// TIA Portal V19 export
FUNCTION_BLOCK "Losma_FB"   // FB154, LAD
TITLE = MATERIAL LUBRICATION (LOSMA)
// stored: MemoryReserve 100, SetENOAutomatically false
   VAR_INPUT
      AreaInterface : "AreaInterface";
      ZSI : "udt_ZoneSafetyInterface";
      DSI : "udt_DeviceSafetyInterface";
      DataIn : Struct
         PbPumpStop : Bool;
         PbPumpStart : Bool;
         PbBlowerStop : Bool;
         PbBlowerStart : Bool;
         PbOilSeparatorStop : Bool;
         PbOilSeparatorStart : Bool;
         SensorLevelTank : Bool;
         SensorStartCloth : Bool;
         SensorOilSeparator : Bool;
         PumpFdbkRunning : Bool;
         OilSeparatorFdbkRunning : Bool;
         ClothFdbkRunning : Bool;
      END_STRUCT;
      CIn : Struct
         EnableStopInPhase : Bool;
         EnableStopProgrammed : Bool;
         EnableAborting : Bool;
         MaterialMoving : Bool;
      END_STRUCT;
      Config : Struct
         EnableWngSystemOff : Bool;
         ClothExist : Bool;
         OilSeparatorExist : Bool;
         LowTankLevelDly : Time;
      END_STRUCT;
   END_VAR
   VAR_OUTPUT
      MachineInterface : "MachineInterface";
      DataOut : Struct
         KmPump : Bool;
         KmCloth : Bool;
         KmOilSeparator : Bool;
         BlowerSolenoidValve : Bool;
         PumpLamp : Bool;
         BlowerLamp : Bool;
      END_STRUCT;
      COut : Struct
         PumpIsRunning : Bool;
         BlowerIsRunning : Bool;
         OilSeparatorIsRunning : Bool;
      END_STRUCT;
   END_VAR
   VAR_IN_OUT
      PersistentValues : Struct
         Par : Struct
            PumpOnOff : Bool;
            BlowerOnOff : Bool;
            OilSeparator : Bool;
            PumpDelayOff : Time;
            BlowerDelayOff : Time;
         END_STRUCT;
      END_STRUCT;
   END_VAR
   VAR
      Sts : Struct
         AlarmsPresence : Bool;
         WarningsPresence : Bool;
         IsStandstill : Bool;
         PumpRunReq : Bool;
         BlowerRunReq : Bool;
         OilSeparatorRunReq : Bool;
         CndPump { ExternalAccessible := 'False'; ExternalVisible := 'False'; ExternalWritable := 'False'} : Bool;
         CndBlower { ExternalAccessible := 'False'; ExternalVisible := 'False'; ExternalWritable := 'False'} : Bool;
         CndCloth { ExternalAccessible := 'False'; ExternalVisible := 'False'; ExternalWritable := 'False'} : Bool;
         CndOilSeparator : Bool;
      END_STRUCT;
      Ctrl : Struct
         RstAlarms : Bool;
         StopDueDoorOpeningRequest : Bool;
         SafeStop : Bool;
         StopInPhase : Bool;
         StopProgrammed : Bool;
         Pump_ManStart : Bool;
         Pump_AutStart : Bool;
         Blower_ManStart : Bool;
         Blower_AutStart : Bool;
         Cloth_AutStart : Bool;
         OilSeparator_ManStart : Bool;
         OilSeparator_AutStart : Bool;
      END_STRUCT;
      Alr : Struct
         LowTankLevel : Bool;
         HighLevelOilTank : Bool;
         Pump : "MotorAlr";
         Cloth : "MotorAlr";
         OilSeparator : "MotorAlr";
      END_STRUCT;
      Wng : Struct
         NoAutReady : Bool;
         PumpOff : Bool;
         BlowerOff : Bool;
         OilSeparatorOff : Bool;
      END_STRUCT;
      M_Pump : "Motor";
      M_Cloth : "Motor";
      M_OilSeparator : "Motor";
      TON_DelayBlowerStop : IEC_TIMER;
      TON_DelayPumpStop : IEC_TIMER;
      TON_LowTankLevel : IEC_TIMER;
      TON_DelayNoPendingCmd : IEC_TIMER;
      TON_OilTankLevelIsFull : IEC_TIMER;
      PbPumpStart_PEAux : Bool;
      PbBlowerStart_PEAux : Bool;
      PbOilSeparatorStart_PEAux : Bool;
   END_VAR
   VAR_TEMP   // added for the SCL form of the ladder/FBD networks
      _w1 : Bool;
   END_VAR
BEGIN

REGION Network 1 (SCL): Reset alarms command
   #Ctrl.RstAlarms := #AreaInterface.RstAlarms;

   IF  #Ctrl.RstAlarms THEN
       #Wng.NoAutReady := FALSE;
       #Alr.LowTankLevel := FALSE;
       #Alr.HighLevelOilTank := FALSE;
   END_IF;
END_REGION

REGION Network 2: Warning Pump / Blower off
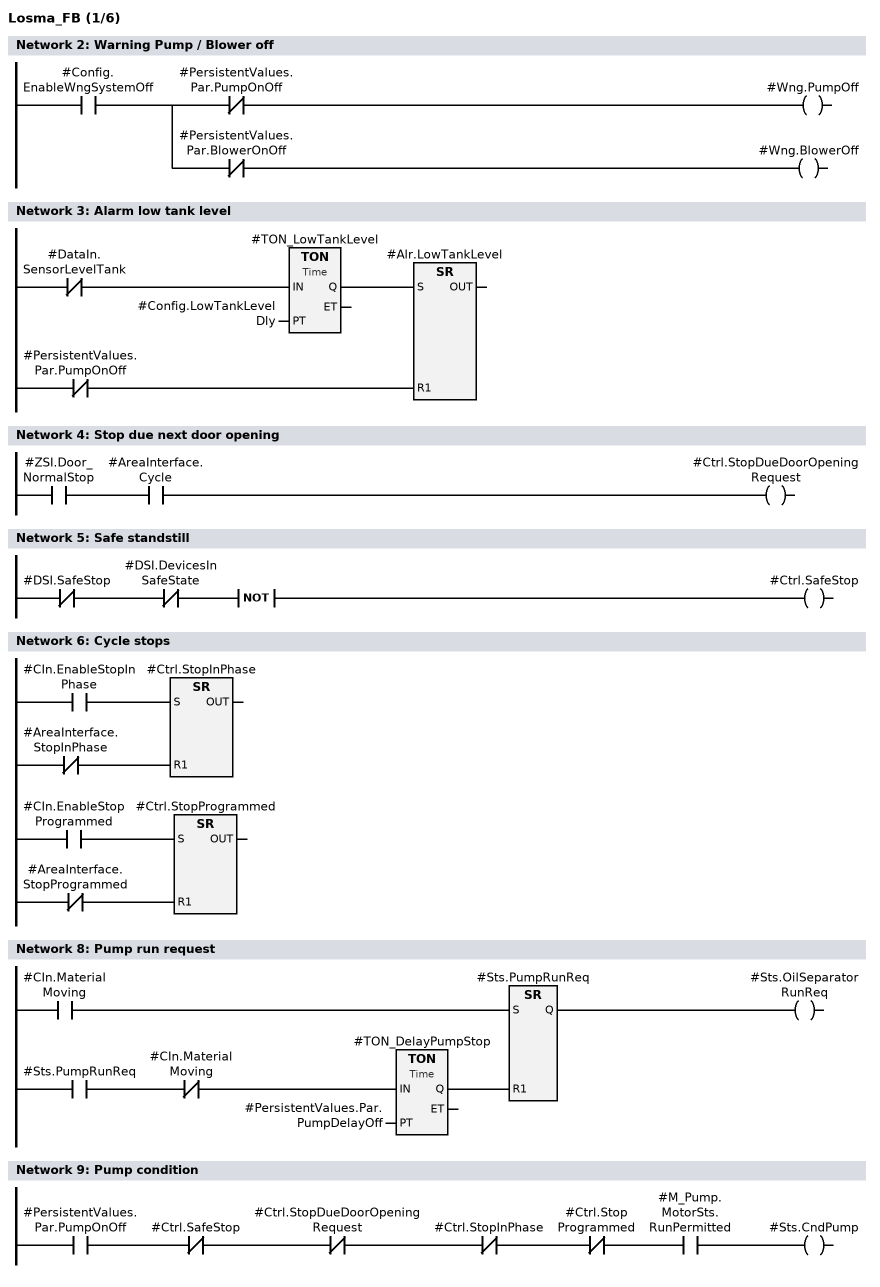
   RUNG wire#powerrail
      Contact( #Config.EnableWngSystemOff )
      wire#w1
      I_Contact( #PersistentValues.Par.PumpOnOff )
      Coil( #Wng.PumpOff )
   END_RUNG
   RUNG wire#w1
      I_Contact( #PersistentValues.Par.BlowerOnOff )
      Coil( #Wng.BlowerOff )
   END_RUNG
   // the same network as SCL:
   #Wng.PumpOff := #Config.EnableWngSystemOff AND NOT #PersistentValues.Par.PumpOnOff;
   #Wng.BlowerOff := #Config.EnableWngSystemOff AND NOT #PersistentValues.Par.BlowerOnOff;
END_REGION

REGION Network 3: Alarm low tank level
   RUNG wire#powerrail
      I_Contact( #DataIn.SensorLevelTank )
      { S7_Templates := "time_type := Time" } #TON_LowTankLevel.TON(pt := #Config.LowTankLevelDly, et =>)
      S_SR(operand := #Alr.LowTankLevel, r1 := wire#w1)
   END_RUNG
   RUNG wire#powerrail
      I_Contact( #PersistentValues.Par.PumpOnOff )
   END_RUNG wire#w1
   // the same network as SCL:
   #TON_LowTankLevel.TON(IN := NOT #DataIn.SensorLevelTank, PT := #Config.LowTankLevelDly);
   IF #TON_LowTankLevel.Q THEN
       #Alr.LowTankLevel := TRUE;   // SR flip-flop
   END_IF;
   IF NOT #PersistentValues.Par.PumpOnOff THEN #Alr.LowTankLevel := FALSE; END_IF;
END_REGION

REGION Network 4: Stop due next door opening
   RUNG wire#powerrail
      Contact( #ZSI.Door_NormalStop )
      Contact( #AreaInterface.Cycle )
      Coil( #Ctrl.StopDueDoorOpeningRequest )
   END_RUNG
   // the same network as SCL:
   #Ctrl.StopDueDoorOpeningRequest := #ZSI.Door_NormalStop AND #AreaInterface.Cycle;
END_REGION

REGION Network 5: Safe standstill
   RUNG wire#powerrail
      I_Contact( #DSI.SafeStop )
      I_Contact( #DSI.DevicesInSafeState )
      Not()
      Coil( #Ctrl.SafeStop )
   END_RUNG
   // the same network as SCL:
   #Ctrl.SafeStop := NOT (NOT #DSI.SafeStop AND NOT #DSI.DevicesInSafeState);
END_REGION

REGION Network 6: Cycle stops
   RUNG wire#powerrail
      Contact( #CIn.EnableStopInPhase )
      S_SR(operand := #Ctrl.StopInPhase, r1 := wire#w1)
   END_RUNG
   RUNG wire#powerrail
      I_Contact( #AreaInterface.StopInPhase )
   END_RUNG wire#w1
   RUNG wire#powerrail
      Contact( #CIn.EnableStopProgrammed )
      S_SR(operand := #Ctrl.StopProgrammed, r1 := wire#w2)
   END_RUNG
   RUNG wire#powerrail
      I_Contact( #AreaInterface.StopProgrammed )
   END_RUNG wire#w2
   // the same network as SCL:
   IF #CIn.EnableStopInPhase THEN
       #Ctrl.StopInPhase := TRUE;   // SR flip-flop
   END_IF;
   IF NOT #AreaInterface.StopInPhase THEN #Ctrl.StopInPhase := FALSE; END_IF;
   IF #CIn.EnableStopProgrammed THEN
       #Ctrl.StopProgrammed := TRUE;   // SR flip-flop
   END_IF;
   IF NOT #AreaInterface.StopProgrammed THEN #Ctrl.StopProgrammed := FALSE; END_IF;
END_REGION

REGION Network 7: <<< PUMP >>>
END_REGION

REGION Network 8: Pump run request
   RUNG wire#powerrail
      Contact( #CIn.MaterialMoving )
      S_SR(operand := #Sts.PumpRunReq, r1 := wire#w1)
      Coil( #Sts.OilSeparatorRunReq )
   END_RUNG
   RUNG wire#powerrail
      Contact( #Sts.PumpRunReq )
      I_Contact( #CIn.MaterialMoving )
      { S7_Templates := "time_type := Time" } #TON_DelayPumpStop.TON(pt := #PersistentValues.Par.PumpDelayOff, et =>)
   END_RUNG wire#w1
   // the same network as SCL:
   #TON_DelayPumpStop.TON(IN := #Sts.PumpRunReq AND NOT #CIn.MaterialMoving,
                          PT := #PersistentValues.Par.PumpDelayOff);
   IF #CIn.MaterialMoving THEN
       #Sts.PumpRunReq := TRUE;   // SR flip-flop
   END_IF;
   IF #TON_DelayPumpStop.Q THEN #Sts.PumpRunReq := FALSE; END_IF;
   #Sts.OilSeparatorRunReq := #Sts.PumpRunReq;
END_REGION

REGION Network 9: Pump condition
   RUNG wire#powerrail
      Contact( #PersistentValues.Par.PumpOnOff )
      I_Contact( #Ctrl.SafeStop )
      I_Contact( #Ctrl.StopDueDoorOpeningRequest )
      I_Contact( #Ctrl.StopInPhase )
      I_Contact( #Ctrl.StopProgrammed )
      Contact( #M_Pump.MotorSts.RunPermitted )
      Coil( #Sts.CndPump )
   END_RUNG
   // the same network as SCL:
   #Sts.CndPump := #PersistentValues.Par.PumpOnOff AND NOT #Ctrl.SafeStop AND NOT #Ctrl.StopDueDoorOpeningRequest AND NOT #Ctrl.StopInPhase AND NOT #Ctrl.StopProgrammed AND #M_Pump.MotorSts.RunPermitted;
END_REGION

REGION Network 10: Pump automatic start
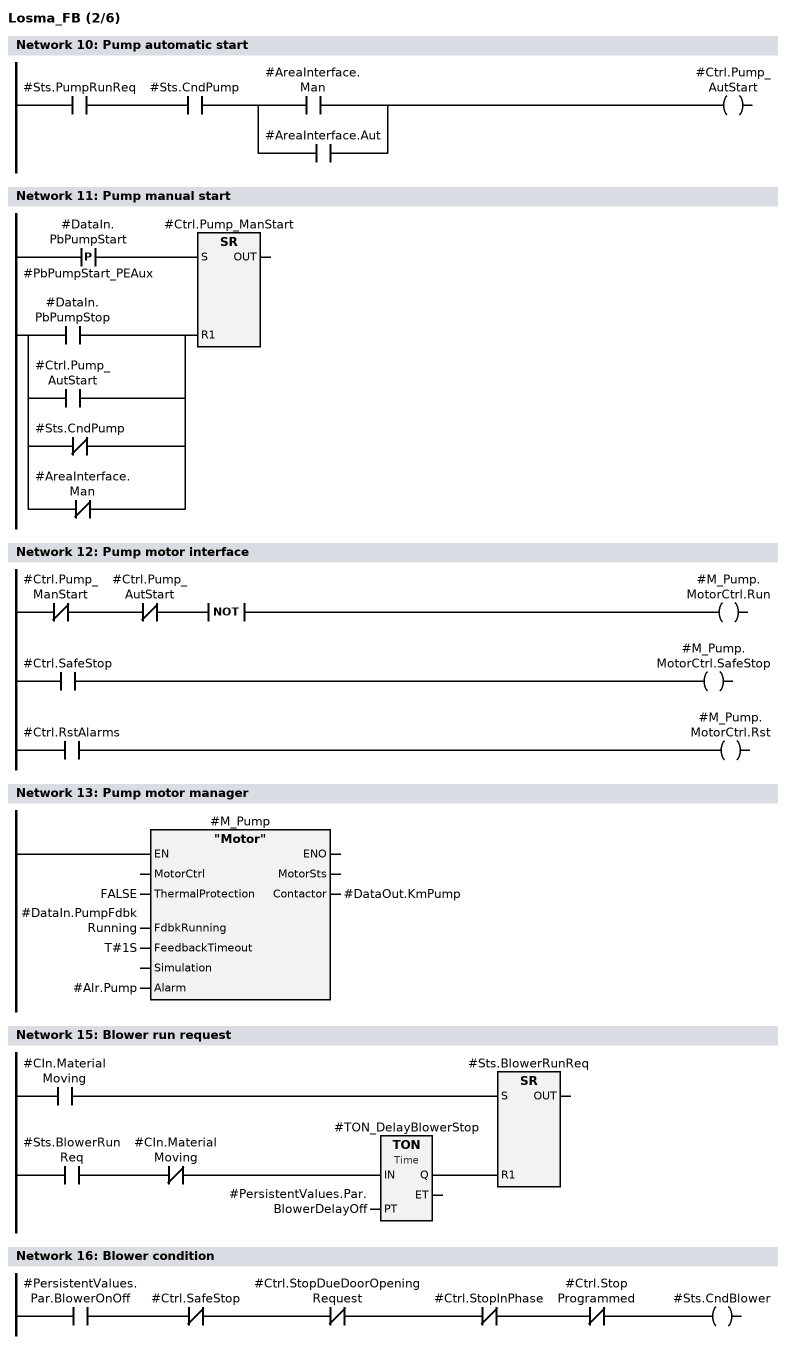
   RUNG wire#powerrail
      Contact( #Sts.PumpRunReq )
      Contact( #Sts.CndPump )
      wire#w1
      Contact( #AreaInterface.Man )
      wire#w2
      Coil( #Ctrl.Pump_AutStart )
   END_RUNG
   RUNG wire#w1
      Contact( #AreaInterface.Aut )
   END_RUNG wire#w2
   // the same network as SCL:
   #Ctrl.Pump_AutStart := #Sts.PumpRunReq AND #Sts.CndPump AND (#AreaInterface.Man OR #AreaInterface.Aut);
END_REGION

REGION Network 11: Pump manual start
   RUNG wire#powerrail
      P_Contact(operand := #DataIn.PbPumpStart, bit := #PbPumpStart_PEAux)
      S_SR(operand := #Ctrl.Pump_ManStart, r1 := wire#w1)
   END_RUNG
   RUNG wire#powerrail
      Contact( #DataIn.PbPumpStop )
   END_RUNG wire#w1
   RUNG wire#powerrail
      Contact( #Ctrl.Pump_AutStart )
   END_RUNG wire#w1
   RUNG wire#powerrail
      I_Contact( #Sts.CndPump )
   END_RUNG wire#w1
   RUNG wire#powerrail
      I_Contact( #AreaInterface.Man )
   END_RUNG wire#w1
   // the same network as SCL:
   #_w1 := #DataIn.PbPumpStart AND NOT #PbPumpStart_PEAux;   // rising edge of #DataIn.PbPumpStart
   #PbPumpStart_PEAux := #DataIn.PbPumpStart;
   IF #_w1 THEN
       #Ctrl.Pump_ManStart := TRUE;   // SR flip-flop
   END_IF;
   IF #DataIn.PbPumpStop OR #Ctrl.Pump_AutStart OR NOT #Sts.CndPump OR NOT #AreaInterface.Man THEN
       #Ctrl.Pump_ManStart := FALSE;
   END_IF;
END_REGION

REGION Network 12: Pump motor interface
   RUNG wire#powerrail
      I_Contact( #Ctrl.Pump_ManStart )
      I_Contact( #Ctrl.Pump_AutStart )
      Not()
      Coil( #M_Pump.MotorCtrl.Run )
   END_RUNG
   RUNG wire#powerrail
      Contact( #Ctrl.SafeStop )
      Coil( #M_Pump.MotorCtrl.SafeStop )
   END_RUNG
   RUNG wire#powerrail
      Contact( #Ctrl.RstAlarms )
      Coil( #M_Pump.MotorCtrl.Rst )
   END_RUNG
   // the same network as SCL:
   #M_Pump.MotorCtrl.Run := NOT (NOT #Ctrl.Pump_ManStart AND NOT #Ctrl.Pump_AutStart);
   #M_Pump.MotorCtrl.SafeStop := #Ctrl.SafeStop;
   #M_Pump.MotorCtrl.Rst := #Ctrl.RstAlarms;
END_REGION

REGION Network 13: Pump motor manager
   RUNG wire#powerrail
      #M_Pump(MotorCtrl :=, ThermalProtection := FALSE, FdbkRunning := #DataIn.PumpFdbkRunning, FeedbackTimeout := T#1S, Simulation :=, Alarm := #Alr.Pump, MotorSts =>, Contactor => #DataOut.KmPump)
   END_RUNG
   // the same network as SCL:
   #M_Pump(ThermalProtection := FALSE,   // "Motor"
           FdbkRunning := #DataIn.PumpFdbkRunning,
           FeedbackTimeout := T#1S,
           Alarm := #Alr.Pump,
           Contactor => #DataOut.KmPump);
END_REGION

REGION Network 14: <<< BLOWER >>>
END_REGION

REGION Network 15: Blower run request
   RUNG wire#powerrail
      Contact( #CIn.MaterialMoving )
      S_SR(operand := #Sts.BlowerRunReq, r1 := wire#w1)
   END_RUNG
   RUNG wire#powerrail
      Contact( #Sts.BlowerRunReq )
      I_Contact( #CIn.MaterialMoving )
      { S7_Templates := "time_type := Time" } #TON_DelayBlowerStop.TON(pt := #PersistentValues.Par.BlowerDelayOff, et =>)
   END_RUNG wire#w1
   // the same network as SCL:
   #TON_DelayBlowerStop.TON(IN := #Sts.BlowerRunReq AND NOT #CIn.MaterialMoving,
                           PT := #PersistentValues.Par.BlowerDelayOff);
   IF #CIn.MaterialMoving THEN
       #Sts.BlowerRunReq := TRUE;   // SR flip-flop
   END_IF;
   IF #TON_DelayBlowerStop.Q THEN #Sts.BlowerRunReq := FALSE; END_IF;
END_REGION

REGION Network 16: Blower condition
   RUNG wire#powerrail
      Contact( #PersistentValues.Par.BlowerOnOff )
      I_Contact( #Ctrl.SafeStop )
      I_Contact( #Ctrl.StopDueDoorOpeningRequest )
      I_Contact( #Ctrl.StopInPhase )
      I_Contact( #Ctrl.StopProgrammed )
      Coil( #Sts.CndBlower )
   END_RUNG
   // the same network as SCL:
   #Sts.CndBlower := #PersistentValues.Par.BlowerOnOff AND NOT #Ctrl.SafeStop AND NOT #Ctrl.StopDueDoorOpeningRequest AND NOT #Ctrl.StopInPhase AND NOT #Ctrl.StopProgrammed;
END_REGION

REGION Network 17: Blower automatc start / blower automatc start
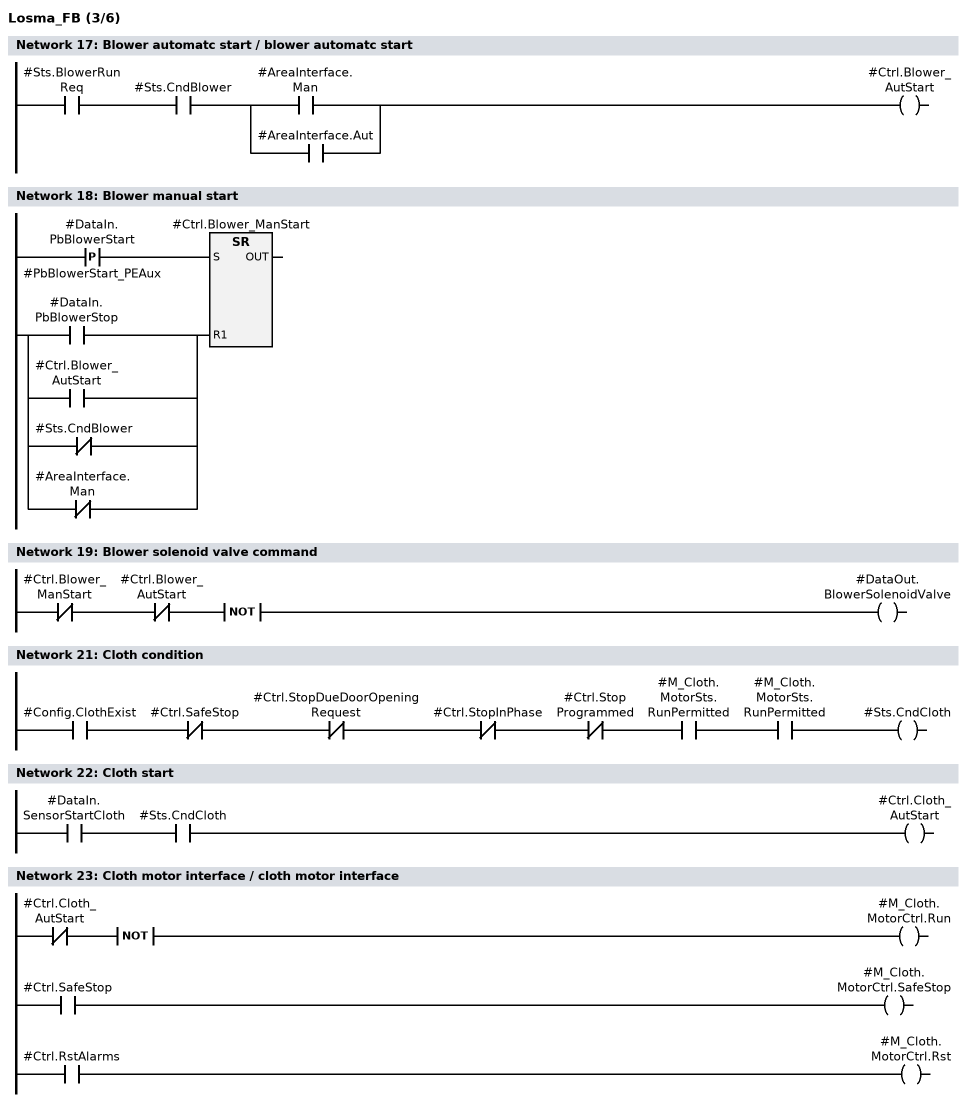
   RUNG wire#powerrail
      Contact( #Sts.BlowerRunReq )
      Contact( #Sts.CndBlower )
      wire#w1
      Contact( #AreaInterface.Man )
      wire#w2
      Coil( #Ctrl.Blower_AutStart )
   END_RUNG
   RUNG wire#w1
      Contact( #AreaInterface.Aut )
   END_RUNG wire#w2
   // the same network as SCL:
   #Ctrl.Blower_AutStart := #Sts.BlowerRunReq AND #Sts.CndBlower AND (#AreaInterface.Man OR #AreaInterface.Aut);
END_REGION

REGION Network 18: Blower manual start
   RUNG wire#powerrail
      P_Contact(operand := #DataIn.PbBlowerStart, bit := #PbBlowerStart_PEAux)
      S_SR(operand := #Ctrl.Blower_ManStart, r1 := wire#w1)
   END_RUNG
   RUNG wire#powerrail
      Contact( #DataIn.PbBlowerStop )
   END_RUNG wire#w1
   RUNG wire#powerrail
      Contact( #Ctrl.Blower_AutStart )
   END_RUNG wire#w1
   RUNG wire#powerrail
      I_Contact( #Sts.CndBlower )
   END_RUNG wire#w1
   RUNG wire#powerrail
      I_Contact( #AreaInterface.Man )
   END_RUNG wire#w1
   // the same network as SCL:
   #_w1 := #DataIn.PbBlowerStart AND NOT #PbBlowerStart_PEAux;   // rising edge of #DataIn.PbBlowerStart
   #PbBlowerStart_PEAux := #DataIn.PbBlowerStart;
   IF #_w1 THEN
       #Ctrl.Blower_ManStart := TRUE;   // SR flip-flop
   END_IF;
   IF #DataIn.PbBlowerStop OR #Ctrl.Blower_AutStart OR NOT #Sts.CndBlower OR NOT #AreaInterface.Man THEN
       #Ctrl.Blower_ManStart := FALSE;
   END_IF;
END_REGION

REGION Network 19: Blower solenoid valve command
   RUNG wire#powerrail
      I_Contact( #Ctrl.Blower_ManStart )
      I_Contact( #Ctrl.Blower_AutStart )
      Not()
      Coil( #DataOut.BlowerSolenoidValve )
   END_RUNG
   // the same network as SCL:
   #DataOut.BlowerSolenoidValve := NOT (NOT #Ctrl.Blower_ManStart AND NOT #Ctrl.Blower_AutStart);
END_REGION

REGION Network 20: <<< CLOTH >>
END_REGION

REGION Network 21: Cloth condition
   RUNG wire#powerrail
      Contact( #Config.ClothExist )
      I_Contact( #Ctrl.SafeStop )
      I_Contact( #Ctrl.StopDueDoorOpeningRequest )
      I_Contact( #Ctrl.StopInPhase )
      I_Contact( #Ctrl.StopProgrammed )
      Contact( #M_Cloth.MotorSts.RunPermitted )
      Contact( #M_Cloth.MotorSts.RunPermitted )
      Coil( #Sts.CndCloth )
   END_RUNG
   // the same network as SCL:
   #Sts.CndCloth := #Config.ClothExist AND NOT #Ctrl.SafeStop AND NOT #Ctrl.StopDueDoorOpeningRequest AND NOT #Ctrl.StopInPhase AND NOT #Ctrl.StopProgrammed AND #M_Cloth.MotorSts.RunPermitted AND #M_Cloth.MotorSts.RunPermitted;
END_REGION

REGION Network 22: Cloth start
   RUNG wire#powerrail
      Contact( #DataIn.SensorStartCloth )
      Contact( #Sts.CndCloth )
      Coil( #Ctrl.Cloth_AutStart )
   END_RUNG
   // the same network as SCL:
   #Ctrl.Cloth_AutStart := #DataIn.SensorStartCloth AND #Sts.CndCloth;
END_REGION

REGION Network 23: Cloth motor interface / cloth motor interface
   RUNG wire#powerrail
      I_Contact( #Ctrl.Cloth_AutStart )
      Not()
      Coil( #M_Cloth.MotorCtrl.Run )
   END_RUNG
   RUNG wire#powerrail
      Contact( #Ctrl.SafeStop )
      Coil( #M_Cloth.MotorCtrl.SafeStop )
   END_RUNG
   RUNG wire#powerrail
      Contact( #Ctrl.RstAlarms )
      Coil( #M_Cloth.MotorCtrl.Rst )
   END_RUNG
   // the same network as SCL:
   #M_Cloth.MotorCtrl.Run := NOT (NOT #Ctrl.Cloth_AutStart);
   #M_Cloth.MotorCtrl.SafeStop := #Ctrl.SafeStop;
   #M_Cloth.MotorCtrl.Rst := #Ctrl.RstAlarms;
END_REGION

REGION Network 24: Cloth motor manager / cloth motor manager
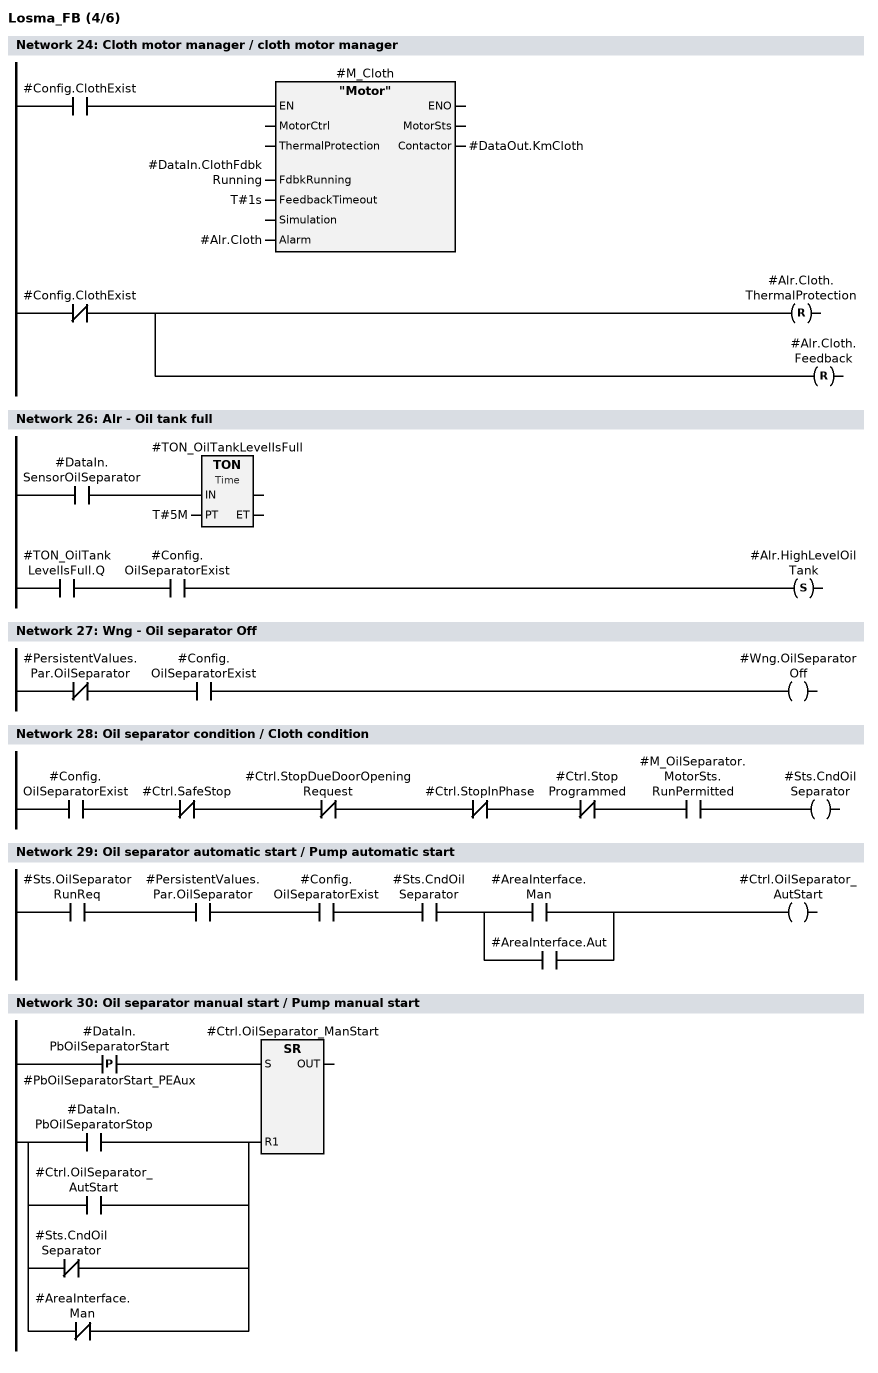
   RUNG wire#powerrail
      Contact( #Config.ClothExist )
      #M_Cloth(MotorCtrl :=, ThermalProtection :=, FdbkRunning := #DataIn.ClothFdbkRunning, FeedbackTimeout := T#1s, Simulation :=, Alarm := #Alr.Cloth, MotorSts =>, Contactor => #DataOut.KmCloth)
   END_RUNG
   RUNG wire#powerrail
      I_Contact( #Config.ClothExist )
      wire#w1
      R_Coil( #Alr.Cloth.ThermalProtection )
   END_RUNG
   RUNG wire#w1
      R_Coil( #Alr.Cloth.Feedback )
   END_RUNG
   // the same network as SCL:
   IF #Config.ClothExist THEN
       #M_Cloth(FdbkRunning := #DataIn.ClothFdbkRunning,   // "Motor"
                FeedbackTimeout := T#1s,
                Alarm := #Alr.Cloth,
                Contactor => #DataOut.KmCloth);
   END_IF;
   IF NOT #Config.ClothExist THEN
       #Alr.Cloth.ThermalProtection := FALSE;
       #Alr.Cloth.Feedback := FALSE;
   END_IF;
END_REGION

REGION Network 25: <<< OIL SEPARATOR >> / <<< CLOTH >>
END_REGION

REGION Network 26: Alr - Oil tank full
   RUNG wire#powerrail
      Contact( #DataIn.SensorOilSeparator )
      { S7_Templates := "time_type := Time" } #TON_OilTankLevelIsFull.TON(pt := T#5M, et =>)
   END_RUNG
   RUNG wire#powerrail
      Contact( #TON_OilTankLevelIsFull.Q )
      Contact( #Config.OilSeparatorExist )
      S_Coil( #Alr.HighLevelOilTank )
   END_RUNG
   // the same network as SCL:
   #TON_OilTankLevelIsFull.TON(IN := #DataIn.SensorOilSeparator, PT := T#5M);
   IF #TON_OilTankLevelIsFull.Q AND #Config.OilSeparatorExist THEN #Alr.HighLevelOilTank := TRUE; END_IF;
END_REGION

REGION Network 27: Wng - Oil separator Off
   RUNG wire#powerrail
      I_Contact( #PersistentValues.Par.OilSeparator )
      Contact( #Config.OilSeparatorExist )
      Coil( #Wng.OilSeparatorOff )
   END_RUNG
   // the same network as SCL:
   #Wng.OilSeparatorOff := NOT #PersistentValues.Par.OilSeparator AND #Config.OilSeparatorExist;
END_REGION

REGION Network 28: Oil separator condition / Cloth condition
   RUNG wire#powerrail
      Contact( #Config.OilSeparatorExist )
      I_Contact( #Ctrl.SafeStop )
      I_Contact( #Ctrl.StopDueDoorOpeningRequest )
      I_Contact( #Ctrl.StopInPhase )
      I_Contact( #Ctrl.StopProgrammed )
      Contact( #M_OilSeparator.MotorSts.RunPermitted )
      Coil( #Sts.CndOilSeparator )
   END_RUNG
   // the same network as SCL:
   #Sts.CndOilSeparator := #Config.OilSeparatorExist AND NOT #Ctrl.SafeStop AND NOT #Ctrl.StopDueDoorOpeningRequest AND NOT #Ctrl.StopInPhase AND NOT #Ctrl.StopProgrammed AND #M_OilSeparator.MotorSts.RunPermitted;
END_REGION

REGION Network 29: Oil separator automatic start / Pump automatic start
   RUNG wire#powerrail
      Contact( #Sts.OilSeparatorRunReq )
      Contact( #PersistentValues.Par.OilSeparator )
      Contact( #Config.OilSeparatorExist )
      Contact( #Sts.CndOilSeparator )
      wire#w1
      Contact( #AreaInterface.Man )
      wire#w2
      Coil( #Ctrl.OilSeparator_AutStart )
   END_RUNG
   RUNG wire#w1
      Contact( #AreaInterface.Aut )
   END_RUNG wire#w2
   // the same network as SCL:
   #Ctrl.OilSeparator_AutStart := #Sts.OilSeparatorRunReq AND #PersistentValues.Par.OilSeparator AND #Config.OilSeparatorExist AND #Sts.CndOilSeparator AND (#AreaInterface.Man OR #AreaInterface.Aut);
END_REGION

REGION Network 30: Oil separator manual start / Pump manual start
   RUNG wire#powerrail
      P_Contact(operand := #DataIn.PbOilSeparatorStart, bit := #PbOilSeparatorStart_PEAux)
      S_SR(operand := #Ctrl.OilSeparator_ManStart, r1 := wire#w1)
   END_RUNG
   RUNG wire#powerrail
      Contact( #DataIn.PbOilSeparatorStop )
   END_RUNG wire#w1
   RUNG wire#powerrail
      Contact( #Ctrl.OilSeparator_AutStart )
   END_RUNG wire#w1
   RUNG wire#powerrail
      I_Contact( #Sts.CndOilSeparator )
   END_RUNG wire#w1
   RUNG wire#powerrail
      I_Contact( #AreaInterface.Man )
   END_RUNG wire#w1
   // the same network as SCL:
   #_w1 := #DataIn.PbOilSeparatorStart AND NOT #PbOilSeparatorStart_PEAux;   // rising edge of #DataIn.PbOilSeparatorStart
   #PbOilSeparatorStart_PEAux := #DataIn.PbOilSeparatorStart;
   IF #_w1 THEN
       #Ctrl.OilSeparator_ManStart := TRUE;   // SR flip-flop
   END_IF;
   IF #DataIn.PbOilSeparatorStop OR #Ctrl.OilSeparator_AutStart OR NOT #Sts.CndOilSeparator OR NOT #AreaInterface.Man THEN
       #Ctrl.OilSeparator_ManStart := FALSE;
   END_IF;
END_REGION

REGION Network 31: Oil separator motor interface / cloth motor interface
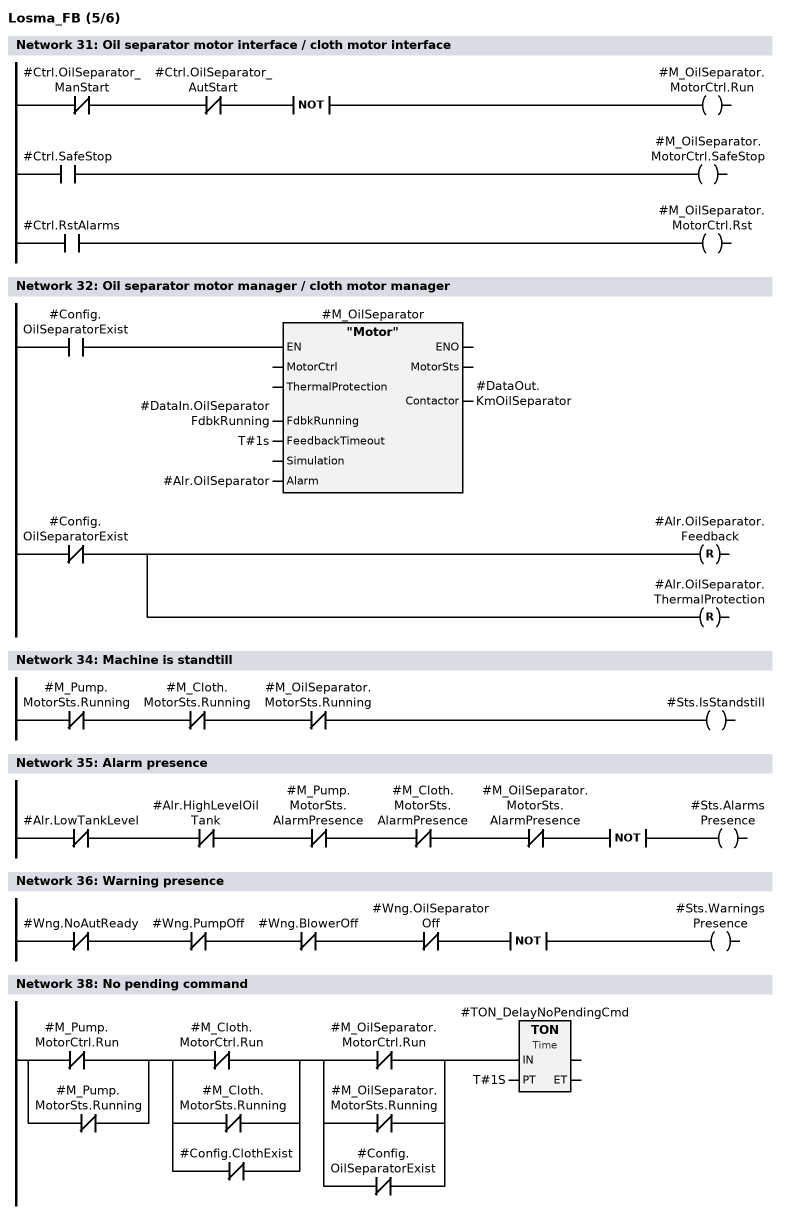
   RUNG wire#powerrail
      I_Contact( #Ctrl.OilSeparator_ManStart )
      I_Contact( #Ctrl.OilSeparator_AutStart )
      Not()
      Coil( #M_OilSeparator.MotorCtrl.Run )
   END_RUNG
   RUNG wire#powerrail
      Contact( #Ctrl.SafeStop )
      Coil( #M_OilSeparator.MotorCtrl.SafeStop )
   END_RUNG
   RUNG wire#powerrail
      Contact( #Ctrl.RstAlarms )
      Coil( #M_OilSeparator.MotorCtrl.Rst )
   END_RUNG
   // the same network as SCL:
   #M_OilSeparator.MotorCtrl.Run := NOT (NOT #Ctrl.OilSeparator_ManStart AND NOT #Ctrl.OilSeparator_AutStart);
   #M_OilSeparator.MotorCtrl.SafeStop := #Ctrl.SafeStop;
   #M_OilSeparator.MotorCtrl.Rst := #Ctrl.RstAlarms;
END_REGION

REGION Network 32: Oil separator motor manager / cloth motor manager
   RUNG wire#powerrail
      Contact( #Config.OilSeparatorExist )
      #M_OilSeparator(MotorCtrl :=, ThermalProtection :=, FdbkRunning := #DataIn.OilSeparatorFdbkRunning, FeedbackTimeout := T#1s, Simulation :=, Alarm := #Alr.OilSeparator, MotorSts =>, Contactor => #DataOut.KmOilSeparator)
   END_RUNG
   RUNG wire#powerrail
      I_Contact( #Config.OilSeparatorExist )
      wire#w1
      R_Coil( #Alr.OilSeparator.Feedback )
   END_RUNG
   RUNG wire#w1
      R_Coil( #Alr.OilSeparator.ThermalProtection )
   END_RUNG
   // the same network as SCL:
   IF #Config.OilSeparatorExist THEN
       #M_OilSeparator(FdbkRunning := #DataIn.OilSeparatorFdbkRunning,   // "Motor"
                       FeedbackTimeout := T#1s,
                       Alarm := #Alr.OilSeparator,
                       Contactor => #DataOut.KmOilSeparator);
   END_IF;
   IF NOT #Config.OilSeparatorExist THEN
       #Alr.OilSeparator.Feedback := FALSE;
       #Alr.OilSeparator.ThermalProtection := FALSE;
   END_IF;
END_REGION

REGION Network 33: <<< >>>
END_REGION

REGION Network 34: Machine is standtill
   RUNG wire#powerrail
      I_Contact( #M_Pump.MotorSts.Running )
      I_Contact( #M_Cloth.MotorSts.Running )
      I_Contact( #M_OilSeparator.MotorSts.Running )
      Coil( #Sts.IsStandstill )
   END_RUNG
   // the same network as SCL:
   #Sts.IsStandstill := NOT #M_Pump.MotorSts.Running AND NOT #M_Cloth.MotorSts.Running AND NOT #M_OilSeparator.MotorSts.Running;
END_REGION

REGION Network 35: Alarm presence
   RUNG wire#powerrail
      I_Contact( #Alr.LowTankLevel )
      I_Contact( #Alr.HighLevelOilTank )
      I_Contact( #M_Pump.MotorSts.AlarmPresence )
      I_Contact( #M_Cloth.MotorSts.AlarmPresence )
      I_Contact( #M_OilSeparator.MotorSts.AlarmPresence )
      Not()
      Coil( #Sts.AlarmsPresence )
   END_RUNG
   // the same network as SCL:
   #Sts.AlarmsPresence := NOT (NOT #Alr.LowTankLevel AND NOT #Alr.HighLevelOilTank AND NOT #M_Pump.MotorSts.AlarmPresence AND NOT #M_Cloth.MotorSts.AlarmPresence AND NOT #M_OilSeparator.MotorSts.AlarmPresence);
END_REGION

REGION Network 36: Warning presence
   RUNG wire#powerrail
      I_Contact( #Wng.NoAutReady )
      I_Contact( #Wng.PumpOff )
      I_Contact( #Wng.BlowerOff )
      I_Contact( #Wng.OilSeparatorOff )
      Not()
      Coil( #Sts.WarningsPresence )
   END_RUNG
   // the same network as SCL:
   #Sts.WarningsPresence := NOT (NOT #Wng.NoAutReady AND NOT #Wng.PumpOff AND NOT #Wng.BlowerOff AND NOT #Wng.OilSeparatorOff);
END_REGION

REGION Network 37 (SCL): Collect machine to area interface
   // Status machine ready
   #MachineInterface.AutReady := #AreaInterface.Aut AND NOT #Sts.AlarmsPresence;
   // Status machine aborting
   #MachineInterface.Aborting := #Sts.AlarmsPresence;
   // Status Ack Stop in phase
   #MachineInterface.AckStopInPhase := #Ctrl.StopInPhase AND #MachineInterface.MotionsStandStill;
   // Status Ack Stop programmed
   #MachineInterface.AckStopProgrammed := #Ctrl.StopProgrammed AND #MachineInterface.MotionsStandStill;
   // Status Motion standtill
   #MachineInterface.MotionsStandStill := #Sts.IsStandstill;
   // Status Alarm presence
   #MachineInterface.AlarmsPresence := #Sts.AlarmsPresence;
   // Status Warning presence
   #MachineInterface.WarningPresence := #Sts.WarningsPresence;

   // Warning machine not automatic ready
   IF #AreaInterface.CheckAutReady AND NOT #MachineInterface.AutReady THEN
     #Wng.NoAutReady := false;
   END_IF;
END_REGION

REGION Network 38: No pending command
   RUNG wire#powerrail
      I_Contact( #M_Pump.MotorCtrl.Run )
      wire#w1
      I_Contact( #M_Cloth.MotorCtrl.Run )
      wire#w2
      I_Contact( #M_OilSeparator.MotorCtrl.Run )
      wire#w3
      { S7_Templates := "time_type := Time" } #TON_DelayNoPendingCmd.TON(pt := T#1S, et =>)
   END_RUNG
   RUNG wire#powerrail
      I_Contact( #M_Pump.MotorSts.Running )
   END_RUNG wire#w1
   RUNG wire#w1
      I_Contact( #M_Cloth.MotorSts.Running )
   END_RUNG wire#w2
   RUNG wire#w1
      I_Contact( #Config.ClothExist )
   END_RUNG wire#w2
   RUNG wire#w2
      I_Contact( #M_OilSeparator.MotorSts.Running )
   END_RUNG wire#w3
   RUNG wire#w2
      I_Contact( #Config.OilSeparatorExist )
   END_RUNG wire#w3
   // the same network as SCL:
   #TON_DelayNoPendingCmd.TON(IN := (NOT #M_Pump.MotorCtrl.Run OR NOT #M_Pump.MotorSts.Running) AND (NOT #M_Cloth.MotorCtrl.Run OR NOT #M_Cloth.MotorSts.Running OR NOT #Config.ClothExist) AND (NOT #M_OilSeparator.MotorCtrl.Run OR NOT #M_OilSeparator.MotorSts.Running OR NOT #Config.OilSeparatorExist),
                           PT := T#1S);
END_REGION

REGION Network 39: Data Out - Lamps
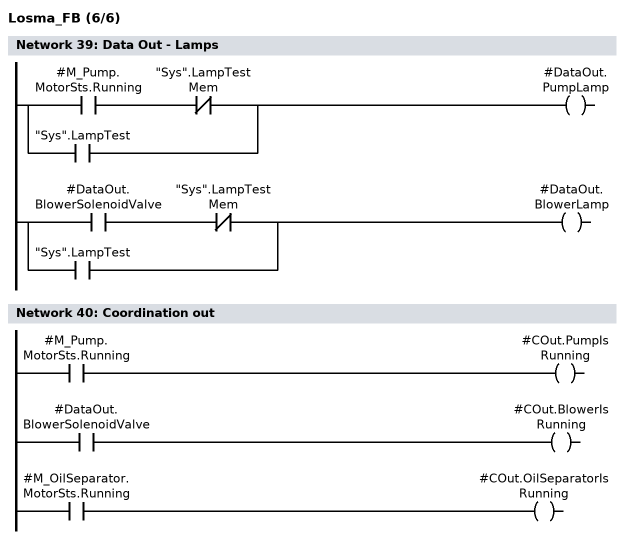
   RUNG wire#powerrail
      Contact( #M_Pump.MotorSts.Running )
      I_Contact( "Sys".LampTestMem )
      wire#w1
      Coil( #DataOut.PumpLamp )
   END_RUNG
   RUNG wire#powerrail
      Contact( "Sys".LampTest )
   END_RUNG wire#w1
   RUNG wire#powerrail
      Contact( #DataOut.BlowerSolenoidValve )
      I_Contact( "Sys".LampTestMem )
      wire#w2
      Coil( #DataOut.BlowerLamp )
   END_RUNG
   RUNG wire#powerrail
      Contact( "Sys".LampTest )
   END_RUNG wire#w2
   // the same network as SCL:
   #DataOut.PumpLamp := (#M_Pump.MotorSts.Running AND NOT "Sys".LampTestMem) OR "Sys".LampTest;
   #DataOut.BlowerLamp := (#DataOut.BlowerSolenoidValve AND NOT "Sys".LampTestMem) OR "Sys".LampTest;
END_REGION

REGION Network 40: Coordination out
   RUNG wire#powerrail
      Contact( #M_Pump.MotorSts.Running )
      Coil( #COut.PumpIsRunning )
   END_RUNG
   RUNG wire#powerrail
      Contact( #DataOut.BlowerSolenoidValve )
      Coil( #COut.BlowerIsRunning )
   END_RUNG
   RUNG wire#powerrail
      Contact( #M_OilSeparator.MotorSts.Running )
      Coil( #COut.OilSeparatorIsRunning )
   END_RUNG
   // the same network as SCL:
   #COut.PumpIsRunning := #M_Pump.MotorSts.Running;
   #COut.BlowerIsRunning := #DataOut.BlowerSolenoidValve;
   #COut.OilSeparatorIsRunning := #M_OilSeparator.MotorSts.Running;
END_REGION
END_FUNCTION_BLOCK
